{attribute 'qualified_only'}
{attribute 'strict'}
TYPE State_Foerderband :
(
	Off,
	Power_up,
	Ready,
	Move_to_next,
	Wait,
	Done,
	Error,
	wait_for_next
);
END_TYPE

(* stored: Version 1.1.0.1, ProductVersion 3.1.4024.12
   DUT State_Foerderband: Id {2c9755a6-4294-4c42-8d9b-84b690300d6c} *)
